{attribute 'qualified_only'}
{attribute 'strict'}
TYPE E_Commands :
(
	noCommand,
	
	//Maint
	calibrate,
	changeAxisEnable,
	changeBrakeState,
	clearAllFaults,
	clearAxisFaults,
	disableAllAxes,
	enableAllAxes,
	goToProd,
	homeAxis,
	moveAxisAbsolute,
	moveAxisRelative,
	turnSafetyOff,
	
	//Prod
	openShutter,
	closeShutter,
	takeExposure,
	
	//Other
	reset
);
END_TYPE

(* stored: Version 1.1.0.1, ProductVersion 3.1.4024.3
   DUT E_Commands: Id {696d3bc0-2295-45ca-96b5-e8fed0b3fbe0} *)
